// TwinCAT 3 PLC project Ring_And_Barrier_System
// ProgramVersion: 3.1.4026.20
// CompilerDefines: VISU_USEPROPERTYINFO
// libraries:
//   Tc2_Standard, * (Beckhoff Automation GmbH)
//   Tc2_System, * (Beckhoff Automation GmbH)
//   Tc2_Utilities, * (Beckhoff Automation GmbH)
// project tree:
//   DUTs/ e_Signal_States.TcDUT, e_Event_Type.TcDUT, e_Street_Type.TcDUT, st_Event.TcDUT, st_Traffic_Phase_Description.TcDUT
//   / GlobalTextList.TcGTLO, PlcTask.TcTTO, Visualization Manager.TcVMO (not stored)
//   GVLs/ Constants.TcGVL, Traffic_Phases.TcGVL
//   POUs/ Check_Phase_Compatibility.TcPOU, fb_CSV_Event_Storage.TcPOU, fb_Event_Buffer.TcPOU, fb_Ring_And_Barrier.TcPOU, fb_Traffic_Phase.TcPOU, i_Persistent_Event_Storage.TcIO, MAIN.TcPOU
//   VISUs/ Initial_Intersection_Visualization.TcVIS
// real-time tasks:
//   TASK PlcTask: cycle T#10ms, priority 20, ADS port 350

CONFIGURATION Ring_And_Barrier_System
    RESOURCE PLC ON TwinCAT3
        TASK PlcTask(INTERVAL := T#10ms, PRIORITY := 20);
        PROGRAM MAIN WITH PlcTask : MAIN;
    END_RESOURCE
END_CONFIGURATION

// ---- DUTs/e_Signal_States.TcDUT
{attribute 'qualified_only'}
{attribute 'strict'}
{attribute 'to_string'}
TYPE e_Signal_States :
(
	ACTIVE_RED := 0,
	ACTIVE_YELLOW := 1,
	ACTIVE_GREEN := 2,
	PASSIVE_RED := 3,
	FLASHING_RED := 4
);
END_TYPE

// ---- DUTs/e_Event_Type.TcDUT
{attribute 'qualified_only'}
{attribute 'strict'}
{attribute 'to_string'}
TYPE e_Event_Type :
(
	Emergency := 0,
	Warning := 1,
	Message := 2,
	Phase_Change := 3
);
END_TYPE

// ---- DUTs/e_Street_Type.TcDUT
{attribute 'qualified_only'}
{attribute 'strict'}
{attribute 'to_string'}
TYPE e_Street_Type :
(
	Major := 0,
	Minor := 1
);
END_TYPE

// ---- DUTs/st_Event.TcDUT
TYPE st_Event :
STRUCT
	e_Event_Type : e_Event_Type;
	e_Event_Severity : TcEventSeverity;
	n_Event_Identity : UDINT;
	s_Event_Text : STRING(255);
	dt_Timestamp : DATE_AND_TIME;
END_STRUCT
END_TYPE

// ---- DUTs/st_Traffic_Phase_Description.TcDUT
TYPE st_Traffic_Phase_Description :
STRUCT
	n_Phase_Identity : UINT;
	e_Street_Identity : e_Street_Type;
	t_Green_Right_Of_Way_Time : TIME;
END_STRUCT
END_TYPE

// ---- GVLs/Constants.TcGVL
{attribute 'qualified_only'}
VAR_GLOBAL CONSTANT
	// The time interval where the yellow light indicates an impending signal change
	t_Yellow_Change_Time : TIME := T#5S;
	
	// The time interval to wait for the intersection to clear before reaching a barrier and starting a new phase
	t_Red_Clearance_Time: TIME := T#3S;
	
	// The time interval for a flashing red signal in the event of a fault
	t_Flashing_Red_Interval : TIME := T#1.5S;
	
	// The time interval alloted for protected left turns
	t_Protected_Left_Turn_Time : TIME := T#5S;
	
	// The time interval alloted for forward travel through the intersection
	t_Forward_Travel_Time : TIME := T#5S;
	
	// The local filepath to the csv event log
	s_CSV_Event_Log_Filepath : T_MaxString := 'C:\Users\Nic C\Documents\twincat3_ws\tc3_Traffic_Light_Project\events.log';
END_VAR

// ---- GVLs/Traffic_Phases.TcGVL
{attribute 'qualified_only'}
VAR_GLOBAL
	// Define the major street traffic phases
	st_Phase_1 : st_Traffic_Phase_Description := (
		n_Phase_Identity := 1,
		e_Street_Identity := e_Street_Type.Major,
		t_Green_Right_Of_Way_Time := Constants.t_Protected_Left_Turn_Time
	);
	
	st_Phase_2 : st_Traffic_Phase_Description := (
		n_Phase_Identity := 2,
		e_Street_Identity := e_Street_Type.Major,
		t_Green_Right_Of_Way_Time := Constants.t_Forward_Travel_Time
	);
	
	st_Phase_5 : st_Traffic_Phase_Description := (
		n_Phase_Identity := 5,
		e_Street_Identity := e_Street_Type.Major,
		t_Green_Right_Of_Way_Time := Constants.t_Protected_Left_Turn_Time
	);
	
	st_Phase_6 : st_Traffic_Phase_Description := (
		n_Phase_Identity := 6,
		e_Street_Identity := e_Street_Type.Major,
		t_Green_Right_Of_Way_Time := Constants.t_Forward_Travel_Time
	);
	
	
	// Define the minor street traffic phases
	st_Phase_3 : st_Traffic_Phase_Description := (
		n_Phase_Identity := 3,
		e_Street_Identity := e_Street_Type.Minor,
		t_Green_Right_Of_Way_Time := Constants.t_Protected_Left_Turn_Time
	);
	
	st_Phase_4 : st_Traffic_Phase_Description := (
		n_Phase_Identity := 4,
		e_Street_Identity := e_Street_Type.Minor,
		t_Green_Right_Of_Way_Time := Constants.t_Forward_Travel_Time
	);
	
	st_Phase_7 : st_Traffic_Phase_Description := (
		n_Phase_Identity := 7,
		e_Street_Identity := e_Street_Type.Minor,
		t_Green_Right_Of_Way_Time := Constants.t_Protected_Left_Turn_Time
	);
	
	st_Phase_8 : st_Traffic_Phase_Description := (
		n_Phase_Identity := 8,
		e_Street_Identity := e_Street_Type.Minor,
		t_Green_Right_Of_Way_Time := Constants.t_Forward_Travel_Time
	);
END_VAR

// ---- POUs/i_Persistent_Event_Storage.TcIO
(*
An interface which can be implemented by various event storage function blocks.
*)

INTERFACE i_Persistent_Event_Storage

METHOD Store_Event
VAR_INPUT
	st_Event_To_Store : st_Event;
END_VAR
END_METHOD

END_INTERFACE

// ---- POUs/MAIN.TcPOU
PROGRAM MAIN
VAR
	// Initialize Major Street Traffic Phase Function Blocks
	fb_Major_Street_Left_Turn_Phase_1 : fb_Traffic_Phase := (st_Phase_Info := Traffic_Phases.st_Phase_1);
	fb_Major_Street_Forward_Phase_2 : fb_Traffic_Phase := (st_Phase_Info := Traffic_Phases.st_Phase_2);
	fb_Major_Street_Left_Turn_Phase_5 : fb_Traffic_Phase := (st_Phase_Info := Traffic_Phases.st_Phase_5);
	fb_Major_Street_Forward_Phase_6 : fb_Traffic_Phase := (st_Phase_Info := Traffic_Phases.st_Phase_6);
	
	// Initialize Minor Street Traffic Phase Function Blocks
	fb_Minor_Street_Left_Turn_Phase_3 : fb_Traffic_Phase := (st_Phase_Info := Traffic_Phases.st_Phase_3);
	fb_Minor_Street_Forward_Phase_4 : fb_Traffic_Phase := (st_Phase_Info := Traffic_Phases.st_Phase_4);
	fb_Minor_Street_Left_Turn_Phase_7 : fb_Traffic_Phase := (st_Phase_Info := Traffic_Phases.st_Phase_7);
	fb_Minor_Street_Forward_Phase_8 : fb_Traffic_Phase := (st_Phase_Info := Traffic_Phases.st_Phase_8);
	
	// Initialize Traffic Phase Arrays
	a_Ring_1 : ARRAY[1..4] OF POINTER TO fb_Traffic_Phase := [
		ADR(fb_Major_Street_Left_Turn_Phase_1),
		ADR(fb_Major_Street_Forward_Phase_2),
		ADR(fb_Minor_Street_Left_Turn_Phase_3),
		ADR(fb_Minor_Street_Forward_Phase_4)
	];
	
	a_Ring_2 : ARRAY[1..4] OF POINTER TO fb_Traffic_Phase := [
		ADR(fb_Major_Street_Left_Turn_Phase_5),
		ADR(fb_Major_Street_Forward_Phase_6),
		ADR(fb_Minor_Street_Left_Turn_Phase_7),
		ADR(fb_Minor_Street_Forward_Phase_8)
	];
	
	// Initialize Traffic Ring Objects
	fb_Ring_One : fb_Ring_And_Barrier := (a_Phase_Sequence := a_Ring_1, fb_Event_Buffer := fb_Event_Buffer);
	fb_Ring_Two : fb_Ring_And_Barrier := (a_Phase_Sequence := a_Ring_2, fb_Event_Buffer := fb_Event_Buffer);
	
	// Initialize the event number for logging
	n_Event_ID : UINT := 1;
	
	// Initialize Event Buffer
	fb_Event_Buffer : fb_Event_Buffer;
	// Initialize Event Read From Buffer
	st_Event_Read_From_Buffer : st_Event;
	// Initialize Error Flag
	b_Error : Bool;
	
	// Initialize CSV Storage
	fb_CSV_Storage : fb_CSV_Event_Storage := (s_Local_File_Path := Constants.s_CSV_Event_Log_Filepath);
	
	// Used to test once
	b_Trigger : BOOL := FALSE;
	fb_Detect_Phase_Complete : F_TRIG;
END_VAR

IF b_Trigger THEN
	fb_Ring_One.Execute_Ring_Sequence(n_Event_ID := n_Event_ID);
	fb_Ring_Two.Execute_Ring_Sequence(n_Event_ID := n_Event_ID);
END_IF

// Call falling edge trigger
fb_Detect_Phase_Complete(CLK := fb_Ring_One.b_Busy);

// Detect a falling edge of the traffic phase being busy
IF fb_Detect_Phase_Complete.Q THEN
	b_Trigger := FALSE;
END_IF

// Write events in buffer if necessary
IF NOT fb_CSV_Storage.b_Busy AND fb_Event_Buffer.n_Events_In_Buffer <> 0 THEN
	fb_Event_Buffer.Get_And_Remove_Event(
		st_Event_Read_From_Buffer => st_Event_Read_From_Buffer,
		b_Error => b_Error
	);
	
	// Store the event in the log
	fb_CSV_Storage.Store_Event(st_Event_To_Store := st_Event_Read_From_Buffer);
END_IF

// Call the storage function block every cycle so that it can continuously logs events
fb_CSV_Storage(s_Local_File_Path := Constants.s_CSV_Event_Log_Filepath);

// Testing flashing stop
//fb_Major_Street_Left_Turn_Phase_1.Flashing_Stop(b_Stop_Traffic := b_Trigger);

END_PROGRAM

// ---- POUs/fb_Traffic_Phase.TcPOU
(*
This function block is used to represent a traffic phase with relevant signal outputs.
*)

FUNCTION_BLOCK fb_Traffic_Phase
// Input phase info struct
VAR_INPUT
	st_Phase_Info : st_Traffic_Phase_Description;
END_VAR

VAR
	// Describes the current active state
	e_State : e_Signal_States := e_Signal_States.PASSIVE_RED;
	
	// Timer for the ACTIVE_GREEN phase
	fb_Green_Signal_Duration : TON;
	
	// Timer for the ACTIVE_YELLOW phase
	fb_Yellow_Signal_Duration : TON;
	
	// Timer for the ACTIVE_RED intersection clearance phase
	fb_Red_Clearance_Signal_Duration : TON;
	
	// Timer for the FLASHING_RED on signal
	fb_Flashing_Red_On_Duration : TON;
	
	// Timer for the FLASHING_RED off signal
	fb_Flashing_Red_Off_Duration : TON;
END_VAR

// Initialize default values for the outputs
VAR_OUTPUT
	b_Green_Signal_Active : BOOL := FALSE;
	b_Yellow_Signal_Active : BOOL := FALSE;
	b_Red_Signal_Active : BOOL := TRUE;
	
	// Describes if the traffic phase is operating
	b_Busy : BOOL := FALSE;
	
	// Output event for logging
	st_Current_Event : st_Event;
END_VAR

METHOD PRIVATE Create_Phase_Event : st_Event
VAR_IN_OUT
	n_Event_ID : UINT;
END_VAR
VAR
	// String of event text
	s_Event_Text : STRING := 'Phase ';
	
	// This allows us to access the PLC system time
	fb_Get_System_Time : GetSystemTime;

	// Create a filetime struct to contain data
	stFileTime : T_FILETIME;
	nLowTime : UDINT;
	nHighTime : UDINT;
	
	// Create a date time object to contain the timestamp
	dt_Timestamp : DT;
END_VAR
VAR_OUTPUT
	st_New_Event : st_Event;
END_VAR
// Define the event ID and increment the count
st_New_Event.n_Event_Identity := n_Event_ID;
n_Event_ID := n_Event_ID + 1;

// Get the current system time from the PLC
fb_Get_System_Time(timeLoDW => nLowTime, timeHiDW => nHighTime);

// Add this information to the filetime struct
stFileTime.dwLowDateTime := nLowTime;
stFileTime.dwHighDateTime := nHighTime;

// Convert this filetime struct to a date time object
dt_Timestamp := FILETIME_TO_DT(fileTime := stFileTime);

// Update the date time in the event struct
st_New_Event.dt_Timestamp := dt_Timestamp;

// Define the event severity
st_New_Event.e_Event_Severity := TcEventSeverity.Verbose;

// Define the event type
st_New_Event.e_Event_Type := e_Event_Type.Phase_Change;

// Define the event text
s_Event_Text := CONCAT(STR1 := s_Event_Text, STR2 := TO_STRING(st_Phase_Info.n_Phase_Identity));
s_Event_Text := CONCAT(STR1 := s_Event_Text, ' ');
s_Event_Text := CONCAT(STR1 := s_Event_Text, STR2 := TO_STRING(e_State));
st_New_Event.s_Event_Text := s_Event_Text;

Create_Phase_Event := st_New_Event;
END_METHOD

(*
Executes the traffic phase with three intervals for ACTIVE_GREEN, ACTIVE_YELLOW, and ACTIVE_RED states.

The input boolean is used to immediately cut short an ACTIVE_GREEN traffic signal in the event of an emergency.
If triggered, the signal switches to ACTIVE_YELLOW then ACTIVE_RED to clear the intersection as soon as possible.
*)

METHOD PUBLIC Excute_Traffic_Phase
VAR_INPUT
	b_Shutdown_Phase_Early : BOOL;
END_VAR
VAR_IN_OUT
	n_Event_ID : UINT;
END_VAR
// This starts the traffic phase
IF NOT b_Busy AND e_State = e_Signal_States.PASSIVE_RED THEN
	// Indicate the traffic phase is operating
	b_Busy := TRUE;
	
	// Advance the state
	e_State := e_Signal_States.ACTIVE_GREEN;
	
	// Create a new event
	st_Current_Event := Create_Phase_Event(n_Event_ID := n_Event_ID);
END_IF

CASE e_State OF
	e_Signal_States.ACTIVE_GREEN:
		// Wait for signal timer to complete or if an early shutdown is triggered
		IF fb_Green_Signal_Duration.Q OR b_Shutdown_Phase_Early THEN
			// Advance the state
			e_State := e_Signal_States.ACTIVE_YELLOW;
			
			// Create a new event
			st_Current_Event := Create_Phase_Event(n_Event_ID := n_Event_ID);
		END_IF
	
		// Define the timer
		fb_Green_Signal_Duration(
			IN := b_Green_Signal_Active AND e_State = e_Signal_States.ACTIVE_GREEN,
			PT := st_Phase_Info.t_Green_Right_Of_Way_Time
		);
	
		// Set the outputs
		b_Green_Signal_Active:= TRUE;
		b_Yellow_Signal_Active := FALSE;
		b_Red_Signal_Active := FALSE;
		
	e_Signal_States.ACTIVE_YELLOW:
		// Wait for signal timer to complete
		IF fb_Yellow_Signal_Duration.Q THEN
			// Advance the state
			e_State := e_Signal_States.ACTIVE_RED;
			
			// Create a new event
			st_Current_Event := Create_Phase_Event(n_Event_ID := n_Event_ID);
		END_IF
		
		// Define the timer
		fb_Yellow_Signal_Duration(
			IN := b_Yellow_Signal_Active AND e_State = e_Signal_States.ACTIVE_YELLOW,
			PT := Constants.t_Yellow_Change_Time
		);
	
		// Set the outputs
		b_Green_Signal_Active:= FALSE;
		b_Yellow_Signal_Active := TRUE;
		b_Red_Signal_Active := FALSE;
		
	e_Signal_States.ACTIVE_RED:
		// Wait for signal timer to complete
		IF fb_Red_Clearance_Signal_Duration.Q THEN
			// Advance the state
			e_State := e_Signal_States.PASSIVE_RED;
		END_IF
		
		// Define the timer
		fb_Red_Clearance_Signal_Duration(
			IN := b_Red_Signal_Active AND e_State = e_Signal_States.ACTIVE_RED,
			PT := Constants.t_Red_Clearance_Time
		);
		
		// Set the outputs
		b_Green_Signal_Active:= FALSE;
		b_Yellow_Signal_Active := FALSE;
		b_Red_Signal_Active := TRUE;
	
	e_Signal_States.PASSIVE_RED:
		// Indicate the traffic phase is not busy
		b_Busy := FALSE;
END_CASE

// Call timers to ensure the elapsed time triggers
fb_Green_Signal_Duration();
fb_Yellow_Signal_Duration();
fb_Red_Clearance_Signal_Duration();
END_METHOD

(*
Signal flashes red indicating traffic must treat the intersection like a stop sign.
*)

METHOD PUBLIC Flashing_Stop
VAR_INPUT
	b_Stop_Traffic : BOOL;
END_VAR
VAR_IN_OUT
	n_Event_ID : UINT;
END_VAR
// Indicate the flashing red phase is operational
IF b_Stop_Traffic AND NOT b_Busy THEN
	// Indicate the phase is busy
	b_Busy := TRUE;
	
	// Set the outputs
	b_Green_Signal_Active:= FALSE;
	b_Yellow_Signal_Active := FALSE;
	
	// Change the state
	e_State := e_Signal_States.FLASHING_RED;
	
	// Create a new event
	st_Current_Event := Create_Phase_Event(n_Event_ID := n_Event_ID);
END_IF

// Input boolean stops this flashing red mode
IF NOT b_Stop_Traffic THEN
	b_Busy := FALSE;
	
	// Stops traffic
	b_Red_Signal_Active := TRUE;
	
	// Change the state
	e_State := e_Signal_States.PASSIVE_RED;
END_IF


// Wait for signal timer to complete
IF fb_Flashing_Red_On_Duration.Q THEN
	// Change the state to flash off
	b_Red_Signal_Active := FALSE;
END_IF

// Wait for signal timer to complete
IF fb_Flashing_Red_Off_Duration.Q THEN
	// Change the state to flash on
	b_Red_Signal_Active := TRUE;
END_IF
	
// Define the timers
fb_Flashing_Red_On_Duration(
	IN := b_Red_Signal_Active AND e_State = e_Signal_States.FLASHING_RED,
	PT := Constants.t_Flashing_Red_Interval
);
fb_Flashing_Red_Off_Duration(
	IN := NOT b_Red_Signal_Active AND e_State = e_Signal_States.FLASHING_RED,
	PT := Constants.t_Flashing_Red_Interval
);

// Call timers to ensure the elapsed time triggers
fb_Flashing_Red_On_Duration();
fb_Flashing_Red_Off_Duration();
END_METHOD

(*
Allows one to adjust the duration of the ACTIVE_GREEN signal.
*)

METHOD PUBLIC Set_Active_Green_Signal_Duration
VAR_INPUT
	t_Input : REFERENCE TO TIME;
END_VAR
st_Phase_Info.t_Green_Right_Of_Way_Time := t_Input;
END_METHOD

END_FUNCTION_BLOCK

// ---- POUs/fb_Ring_And_Barrier.TcPOU
(*
Used to represent the standard ring and barrier sequence for a four way intersection.
*)

FUNCTION_BLOCK fb_Ring_And_Barrier
VAR_INPUT
	a_Phase_Sequence : ARRAY[1..i_Number_Of_Phases] OF POINTER TO fb_Traffic_Phase;
	
	fb_Event_Buffer : REFERENCE TO fb_Event_Buffer;
END_VAR
VAR CONSTANT
	i_Number_Of_Phases : INT := 4;
END_VAR
VAR
	// Trigger to detect the end of a traffic phase
	fb_Detect_Phase_Complete : F_TRIG;
	
	// Index of the traffic phase currently operating in the ring sequence
	i_Ring_Index : INT := 1;
	
	// Used to determine a change in event
	s_Current_Event_Text : STRING(255);;
END_VAR
VAR_OUTPUT
	// Describes if the function block is operating
	b_Busy : BOOL := FALSE;
END_VAR

(*
Executes the standard ring and barrier sequence.
*)

METHOD PUBLIC Execute_Ring_Sequence
VAR_IN_OUT
	n_Event_ID : UINT;
END_VAR
IF NOT b_Busy THEN
	b_Busy := TRUE;
END_IF

// Execute the traffic phase
a_Phase_Sequence[i_Ring_Index]^.Excute_Traffic_Phase(
	n_Event_ID := n_Event_ID,
	b_Shutdown_Phase_Early := FALSE
);

// Detect if a new event is created by the traffic phase function block
IF s_Current_Event_Text <> a_Phase_Sequence[i_Ring_Index]^.st_Current_Event.s_Event_Text THEN
	// Add the event to the buffer
	fb_Event_Buffer.Add_Event(st_Event_To_Add := a_Phase_Sequence[i_Ring_Index]^.st_Current_Event);
	
	// Update the current event text
	s_Current_Event_Text := a_Phase_Sequence[i_Ring_Index]^.st_Current_Event.s_Event_Text;
END_IF

// Call falling edge trigger
fb_Detect_Phase_Complete(CLK := a_Phase_Sequence[i_Ring_Index]^.b_Busy);
	
// Detect if the traffic phase is complete
IF NOT a_Phase_Sequence[i_Ring_Index]^.b_Busy THEN
	// Increment the index
	i_Ring_Index := i_Ring_Index + 1;
	
	// Check if we need to reset the index
	IF i_Ring_Index > i_Number_Of_Phases THEN
		i_Ring_Index := 1;
		
		// Indicate completion
		b_Busy := FALSE;
	END_IF
END_IF
END_METHOD

END_FUNCTION_BLOCK

// ---- POUs/fb_Event_Buffer.TcPOU
(*
FB_EventBuffer is an implementation of an event buffer with the FB_MemRingBuffer function block
provided in the Tc2_Utilities library.
*)

FUNCTION_BLOCK PUBLIC fb_Event_Buffer
VAR
	// Buffer memory used by FB_MemRingBuffer function block
	arr_Buffer_Memory : ARRAY[0..i_Buffer_Memory_Byte_Size] OF BYTE;
	
	// Create an instance of the MemRingBuffer
	fb_Event_Ring_Buffer : FB_MemRingBuffer;
END_VAR

VAR CONSTANT
	// The number of events to store in the event buffer
	i_Number_Of_Events_To_Store_In_Buffer : INT := 10;
	
	// The size of an event in bytes
	i_Event_Byte_Size : INT := SIZEOF(st_Event);
	
	// The total number of bytes in the buffer memory
	i_Buffer_Memory_Byte_Size : INT := i_Number_Of_Events_To_Store_In_Buffer * i_Event_Byte_Size;
END_VAR

VAR_OUTPUT
	n_Events_In_Buffer : UINT := 0;
END_VAR

(*
Attempts to add an event to the buffer and returns a boolean to show if successful.
*)

METHOD PUBLIC Add_Event : BOOL
VAR_INPUT
	st_Event_To_Add : REFERENCE TO st_Event;
END_VAR
VAR_OUTPUT
	b_Error : BOOL;
END_VAR
// Try to add the event to the buffer
fb_Event_Ring_Buffer.A_AddTail(
	pWrite := ADR(st_Event_To_Add),
	cbWrite := SIZEOF(st_Event_To_Add),
	pBuffer := ADR(arr_Buffer_Memory),
	cbBuffer := SIZEOF(arr_Buffer_Memory)
);

// Indicate if successful
b_Error := NOT fb_Event_Ring_Buffer.bOk;

// Increase the count
n_Events_In_Buffer := n_Events_In_Buffer + 1;
END_METHOD

(*
Attemps to read and remove an event from the buffer and returns a boolean to show if successful.
*)

METHOD PUBLIC Get_And_Remove_Event
VAR_OUTPUT
	st_Event_Read_From_Buffer : st_Event;

	b_Error : BOOL;
END_VAR
// Try to read the oldest event from the buffer
fb_Event_Ring_Buffer.A_RemoveHead (
	pRead := ADR(st_Event_Read_From_Buffer),
	cbRead := SIZEOF(st_Event_Read_From_Buffer),
	pBuffer := ADR(arr_Buffer_Memory),
	cbBuffer := SIZEOF(arr_Buffer_Memory)
);

// Indicate if successful
b_Error := NOT fb_Event_Ring_Buffer.bOk;

// Decrease the count
n_Events_In_Buffer := n_Events_In_Buffer - 1;
END_METHOD

(*
Resets the buffer.
*)

METHOD PUBLIC Reset_Buffer : BOOL
VAR_OUTPUT
	b_Error : Bool;
END_VAR
// Reset buffer
fb_Event_Ring_Buffer.A_Reset();

// Indicate if successful
b_Error := NOT fb_Event_Ring_Buffer.bOk;
END_METHOD

END_FUNCTION_BLOCK

// ---- POUs/fb_CSV_Event_Storage.TcPOU
(*
Used to store events in the .csv file format.
*)

FUNCTION_BLOCK fb_CSV_Event_Storage IMPLEMENTS i_Persistent_Event_Storage
VAR_INPUT
	s_Local_File_Path : T_MaxString;
END_VAR

VAR
	e_Write_State : (
		FILE_OPEN_TRIGGER,
		FILE_OPEN,
		WAIT_FOR_EVENT,
		WRITE_EVENT_TRIGGER,
		WRITE_EVENT,
		FILE_CLOSE_TRIGGER,
		FILE_CLOSE,
		ERROR
	);
	
	// Create function blocks to open, write to, and close a csv file
	FB_File_Open : FB_FileOpen;
	FB_File_Write : FB_FilePuts;
	FB_File_Close : FB_FileClose;
	
	// Event to write to csv file
	st_Event_Written_To_File : st_Event;
	
	// String that gets written to the csv file
	s_CSV_String : T_MaxString;
	
	// Error message
	s_Error_Msg : STRING;
END_VAR
VAR_OUTPUT
	b_Busy : BOOL := FALSE; 
	b_Error : BOOL := FALSE;
END_VAR

CASE e_Write_State OF
	FILE_OPEN_TRIGGER:
		FB_File_Open(
			bExecute := TRUE,
			sPathName := s_Local_File_Path,
			nMode := FOPEN_MODEAPPEND
		);
		e_Write_State := FILE_OPEN;
		
		b_Busy := TRUE;
		
	FILE_OPEN :
		FB_File_Open(bExecute := FALSE);
		
		IF FB_File_Open.bError THEN
			e_Write_State := ERROR;
			
			// Write error message
			s_Error_Msg := CONCAT(
				STR1 := 'CSV Event Storage error encountered when opening file with ADS return code of: ',
				STR2 := TO_STRING(FB_File_Close.nErrId)
			);
			
		ELSIF NOT FB_File_Open.bBusy AND FB_File_Open.hfile <> 0 THEN
			e_Write_State := WAIT_FOR_EVENT;
		END_IF
		
	WAIT_FOR_EVENT : 
		b_Busy := FALSE;
		
	WRITE_EVENT_TRIGGER :
		s_CSV_String := Create_CSV_String(st_Event_Data := st_Event_Written_To_File);
		FB_File_Write(
			bExecute := TRUE,
			hFile := FB_File_Open.hFile,
			sLine := s_CSV_String
		);
		e_Write_State := WRITE_EVENT;
		b_Busy := TRUE;
		
	WRITE_EVENT:
		FB_File_Write(bExecute := FALSE);
		
		IF FB_File_Write.bError THEN
			e_Write_State := ERROR;
			
			// Write error message
			s_Error_Msg := CONCAT(
				STR1 := 'CSV Event Storage error encountered when writing to file with ADS return code of: ',
				STR2 := TO_STRING(FB_File_Close.nErrId)
			);
			
		ELSIF NOT FB_File_Write.bBusy THEN
			e_Write_State := WAIT_FOR_EVENT;
		END_IF
	
	FILE_CLOSE_TRIGGER :
		FB_File_Close(
			bExecute := TRUE,
			hFile := FB_File_Open.hFile
		);
		e_Write_State := FILE_CLOSE;
	
	FILE_CLOSE :
		FB_File_Close(bExecute := FALSE);
		
		IF FB_File_Close.bError THEN
			e_Write_State := ERROR;
			
			// Write error message
			s_Error_Msg := CONCAT(
				STR1 := 'CSV Event Storage error encountered when closing file with ADS return code of: ',
				STR2 := TO_STRING(FB_File_Close.nErrId)
			);
			
		ELSIF NOT FB_File_Close.bBusy THEN
			e_Write_State := FILE_OPEN_TRIGGER;
			
		END_IF
		
	ERROR :
		// Write error to log
		ADSLOGSTR(
			msgCtrlMask := ADSLOG_MSGTYPE_ERROR,
			msgFmtStr := s_Error_Msg,
			strArg := ''
		);
		
		b_Error := TRUE;
	
END_CASE

(*
Creates a csv string by concatenating st_Event data
*)

METHOD PRIVATE Create_CSV_String : T_MaxString
VAR_INPUT
	st_Event_Data : REFERENCE TO st_Event;
END_VAR
VAR
	s_Temp_String : STRING(255);
END_VAR
s_Temp_String := TO_STRING(st_Event_Data.n_Event_Identity);
s_Temp_String := CONCAT(STR1 := s_Temp_String, STR2 := ', ');
s_Temp_String := CONCAT(STR1 := s_Temp_String, STR2 := TO_STRING(st_Event_Data.dt_Timestamp));
s_Temp_String := CONCAT(STR1 := s_Temp_String, STR2 := ', ');
s_Temp_String := CONCAT(STR1 := s_Temp_String, STR2 := TO_STRING(st_Event_Data.e_Event_Severity));
s_Temp_String := CONCAT(STR1 := s_Temp_String, STR2 := ', ');
s_Temp_String := CONCAT(STR1 := s_Temp_String, STR2 := TO_STRING(st_Event_Data.e_Event_Type));
s_Temp_String := CONCAT(STR1 := s_Temp_String, STR2 := ', ');
s_Temp_String := CONCAT(STR1 := s_Temp_String, STR2 := st_Event_Data.s_Event_Text);
s_Temp_String := CONCAT(STR1 := s_Temp_String, STR2 := '$n');
Create_CSV_String := s_Temp_String;
END_METHOD

(*
Stores event details in a CSV file
*)
METHOD Store_Event
VAR_INPUT
	st_Event_To_Store : st_Event;
END_VAR
IF e_Write_State = WAIT_FOR_EVENT THEN
	e_Write_State := WRITE_EVENT_TRIGGER;
	
	st_Event_Written_To_File := st_Event_To_Store;
END_IF
END_METHOD

END_FUNCTION_BLOCK

// ---- POUs/Check_Phase_Compatibility.TcPOU
(*
Checks if two traffic phases are compatible using their phase identity number.
Two compatible traffic phases can be run concurrently without causing traffic
conflicts.
*)

FUNCTION Check_Phase_Compatibility : Bool
VAR_INPUT
	fb_Phase_A : REFERENCE TO fb_Traffic_Phase;
	fb_Phase_B : REFERENCE TO fb_Traffic_Phase;
END_VAR
VAR
	n_ID_A : UINT := fb_Phase_A.st_Phase_Info.n_Phase_Identity;
	n_ID_B : UINT := fb_Phase_B.st_Phase_Info.n_Phase_Identity;
END_VAR

// Check the street identity
IF fb_Phase_A.st_Phase_Info.e_Street_Identity = fb_Phase_B.st_Phase_Info.e_Street_Identity THEN
	// Check if one ID is odd and one is even
	IF (n_ID_A + n_ID_B) MOD 2 = 1 THEN
		// If the phase numbers add to 7, meaning we have a 1 + 6 or 2 + 5 pair for the major street
		// or if the phase numbers add to 11, meaning we have a 3 + 8 or 4 + 7 pair for the minor street
		IF (n_ID_A + n_ID_B) = 7 OR (n_ID_A + n_ID_B) = 11 THEN
			Check_Phase_Compatibility := TRUE;
			
		// Other possible configurations are incompatible
		ELSE
			Check_Phase_Compatibility := FALSE;
		END_IF
	
	// IDs are either both odd or both even
	ELSE
		Check_Phase_Compatibility := TRUE;
	END_IF

ELSE
	Check_Phase_Compatibility := FALSE;
END_IF

END_FUNCTION

// ---- GlobalTextList.TcGTLO
TEXTLIST GlobalTextList
  440 = '<=='
  155 = '<==='
  6 = 'Pomerado Rd Northbound'
  65 = 'Pomerado Rd Southbound'
  934 = 'Scripps Poway Pkwy Eastbound'
  475 = 'Scripps Poway Pkwy Westbound'
  348 = '⬅'
END_TEXTLIST

// ---- VISUs/Initial_Intersection_Visualization.TcVIS
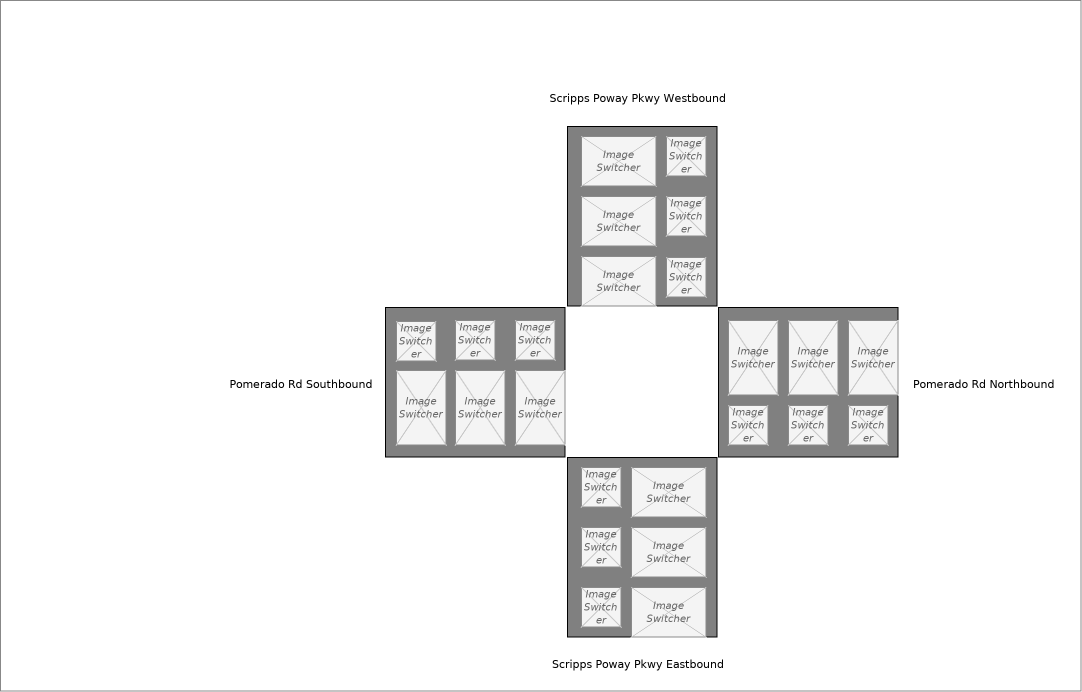
VISUALIZATION Initial_Intersection_Visualization  // 1082x692
    Group (203,71 879x566)
        Group (182,55 513x511)
            Group (182,331 150x180)
                RoundedRectangle (0,0 150x180)
                ImageSwitcher (64,70 75x50), variable: MAIN.fb_Major_Street_Forward_Phase_6.b_Yellow_Signal_Active, behaviour: TOGGLE
                ImageSwitcher (64,130 75x50), variable: MAIN.fb_Major_Street_Forward_Phase_6.b_Green_Signal_Active, behaviour: TOGGLE
                ImageSwitcher (64,10 75x50), variable: MAIN.fb_Major_Street_Forward_Phase_6.b_Red_Signal_Active, behaviour: TOGGLE
                ImageSwitcher (14,10 40x40), variable: MAIN.fb_Major_Street_Left_Turn_Phase_1.b_Red_Signal_Active, behaviour: TOGGLE
                ImageSwitcher (14,70 40x40), variable: MAIN.fb_Major_Street_Left_Turn_Phase_1.b_Yellow_Signal_Active, behaviour: TOGGLE
                ImageSwitcher (14,130 40x40), variable: MAIN.fb_Major_Street_Left_Turn_Phase_1.b_Green_Signal_Active, behaviour: TOGGLE
            Group (333,181 180x150)
                RoundedRectangle (0,0 180x150)
                Group (10,13 170x125)
                    ImageSwitcher (0,0 50x75), variable: MAIN.fb_Minor_Street_Forward_Phase_4.b_Red_Signal_Active, behaviour: TOGGLE
                    ImageSwitcher (60,0 50x75), variable: MAIN.fb_Minor_Street_Forward_Phase_4.b_Yellow_Signal_Active, behaviour: TOGGLE
                    ImageSwitcher (120,0 50x75), variable: MAIN.fb_Minor_Street_Forward_Phase_4.b_Green_Signal_Active, behaviour: TOGGLE
                    ImageSwitcher (0,85 40x40), variable: MAIN.fb_Minor_Street_Left_Turn_Phase_7.b_Red_Signal_Active, behaviour: TOGGLE
                    ImageSwitcher (60,85 40x40), variable: MAIN.fb_Minor_Street_Left_Turn_Phase_7.b_Yellow_Signal_Active, behaviour: TOGGLE
                    ImageSwitcher (120,85 40x40), variable: MAIN.fb_Minor_Street_Left_Turn_Phase_7.b_Green_Signal_Active, behaviour: TOGGLE
            RoundedRectangle (0,181 180x150)
            Group (11,194 169x125)
                ImageSwitcher (119,50 50x75), variable: MAIN.fb_Minor_Street_Forward_Phase_8.b_Red_Signal_Active, behaviour: TOGGLE
                ImageSwitcher (0,50 50x75), variable: MAIN.fb_Minor_Street_Forward_Phase_8.b_Green_Signal_Active, behaviour: TOGGLE
                ImageSwitcher (59,50 50x75), variable: MAIN.fb_Minor_Street_Forward_Phase_8.b_Yellow_Signal_Active, behaviour: TOGGLE
                ImageSwitcher (119,0 40x40), variable: MAIN.fb_Minor_Street_Left_Turn_Phase_3.b_Red_Signal_Active, behaviour: TOGGLE
                ImageSwitcher (59,0 40x40), variable: MAIN.fb_Minor_Street_Left_Turn_Phase_3.b_Yellow_Signal_Active, behaviour: TOGGLE
                ImageSwitcher (0,1 40x40), variable: MAIN.fb_Minor_Street_Left_Turn_Phase_3.b_Green_Signal_Active, behaviour: TOGGLE
            Group (182,0 150x180)
                RoundedRectangle (0,0 150x180)
                Group (14,10 125x170)
                    ImageSwitcher (0,120 75x50), variable: MAIN.fb_Major_Street_Forward_Phase_2.b_Red_Signal_Active, behaviour: TOGGLE
                    ImageSwitcher (0,60 75x50), variable: MAIN.fb_Major_Street_Forward_Phase_2.b_Yellow_Signal_Active, behaviour: TOGGLE
                    ImageSwitcher (0,0 75x50), variable: MAIN.fb_Major_Street_Forward_Phase_2.b_Green_Signal_Active, behaviour: TOGGLE
                    ImageSwitcher (85,121 40x40), variable: MAIN.fb_Major_Street_Left_Turn_Phase_5.b_Red_Signal_Active, behaviour: TOGGLE
                    ImageSwitcher (85,60 40x40), variable: MAIN.fb_Major_Street_Left_Turn_Phase_5.b_Yellow_Signal_Active, behaviour: TOGGLE
                    ImageSwitcher (85,0 40x40), variable: MAIN.fb_Major_Street_Left_Turn_Phase_5.b_Green_Signal_Active, behaviour: TOGGLE
        Label (337,0 196x55), "Scripps Poway Pkwy Westbound"
        Label (683,286 196x55), "Pomerado Rd Northbound"
        Label (0,286 196x55), "Pomerado Rd Southbound"
    Label (540,637 196x55), "Scripps Poway Pkwy Eastbound"
END_VISUALIZATION
